// TwinCAT 3 PLC project SymbolInfo
// ProgramVersion: 3.1.4024.0
// libraries:
//   Tc2_Standard, * (Beckhoff Automation GmbH)
//   Tc2_System, * (Beckhoff Automation GmbH)
//   Tc2_Utilities, * (Beckhoff Automation GmbH)
//   Tc3_Module, * (Beckhoff Automation GmbH)
// project tree:
//   DUTs/ ST_Device.TcDUT
//   GVLs/ Globals.TcGVL
//   / PlcTask.TcTTO (not stored)
//   POUs/ MAIN.TcPOU
// real-time tasks:
//   TASK PlcTask: cycle T#1ms, priority 20, ADS port 350

// ---- DUTs/ST_Device.TcDUT
TYPE ST_Device :
STRUCT
	value : DINT;;
END_STRUCT
END_TYPE

// ---- GVLs/Globals.TcGVL
{attribute 'qualified_only'}
VAR_GLOBAL
	device_1 : ST_Device;
	device_2 : ST_Device;
END_VAR

// ---- POUs/MAIN.TcPOU
PROGRAM MAIN
VAR	
	nState 		    : INT := 0;

	// FBs to get PLC symbol information by symbol's name 
	fbSymbInfo		: PLC_ReadSymInfoByName := ( PORT := 851, TMOUT := DEFAULT_ADS_TIMEOUT );
	stSymbolInfo	: Tc2_Utilities.SYMINFOSTRUCT;

	// FB to change a plc variable by index of group and offset 
	fbWriteReq      : ADSWRITE := ( NETID := '', PORT := 851, TMOUT := DEFAULT_ADS_TIMEOUT );
	
    Variable_Name   : STRING := 'globals.device_1.value';
	Variable_Value  : DINT := 0;	
	
	bFirst			: BOOL := TRUE;
	fbRandom		: DRand;
	
END_VAR

CASE nState OF 

	0:  // reset FB if required
		IF (fbSymbInfo.START AND NOT fbSymbInfo.BUSY) THEN
			fbSymbInfo(START:= FALSE);
		END_IF
		// read symbol information
		fbSymbInfo
    	( 
			symname := 	Variable_Name,
			syminfo => stSymbolInfo,
			start:= TRUE
		);
		// get the result
		IF (fbSymbInfo.BUSY = FALSE) THEN
	 		IF (fbSymbInfo.ERR) THEN
				nState := 99;
			ELSE
				nState := nState +1;
			END_IF
		END_IF
	
	1:	// reset FB if required
		IF (fbWriteReq.WRITE AND NOT fbWriteReq.BUSY) THEN
			fbWriteReq(WRITE:= FALSE);
		END_IF
		// execute write request
		fbWriteReq(
			IDXGRP:= stSymbolInfo.idxGroup, 
			IDXOFFS:= stSymbolInfo.idxOffset, 
			LEN:= stSymbolInfo.byteSize, 
			SRCADDR:= ADR(Variable_Value),
			WRITE := TRUE );
		// get the result
		IF (NOT fbWriteReq.BUSY) THEN
	 		IF (fbWriteReq.ERR) THEN
				nState := 99;
			ELSE
				nState := 100;
			END_IF
		END_IF
	99:
		; // Error
		
	100: // Done
		
		// switch to other variable and apply different value 
		
		IF (bFirst) THEN fbRandom( Seed:= 4711); bFirst:= FALSE; END_IF
		fbRandom();
		Variable_Value := LREAL_TO_DINT (fbRandom.Num * 42);
	
		IF (Variable_Name = 'globals.device_1.value') THEN Variable_Name := 'globals.device_2.value'; END_IF
		
		nState := 0; 

END_CASE

END_PROGRAM
